{attribute 'qualified_only'}
VAR_GLOBAL INTERNAL
END_VAR
VAR_GLOBAL CONSTANT INTERNAL
	fbTcComIecApplicationInfo : FsFB_TcComIecApplicationInfo := ();
END_VAR

(* stored: Version 1.1.0.1, ProductVersion 3.1.4024.4
   GVL _FsGVL: Id {5dda4c9b-0d87-46a8-861c-6a7d19cc7694} *)
